Omron CX-Programmer project NewProject (CX-Programmer 9.61)

# PLC traficlight: CP1E N30

## Global symbols (name address type ; comment)
0.00 BOOL  ; STOP
0.01 BOOL  ; START
0.02 BOOL  ; WAKTU 2
0.05 BOOL  ; SENSOR 1
0.06 BOOL  ; SENSOR 2
100.00 BOOL  ; LAMPU MERAH
100.01 BOOL  ; LAMPU KUNING
100.02 BOOL  ; LAMPU HIJAU
100.03 BOOL  ; LAMPU HIJAU
100.04 BOOL  ; LAMPU KUNING
100.05 BOOL  ; LAMPU MERAH
100.06 BOOL  ; IF
5.00 BOOL  ; IR
5.01 BOOL  ; SENSOR
T001 BOOL  ; WAKTU 1
T002 BOOL  ; WAKTU 2
T003 BOOL  ; WAKTU 3
T004 BOOL  ; WAKTU 4
T005 BOOL  ; WAKTU 5
T006 BOOL  ; WAKTU 2
T007 BOOL  ; WAKTU 6

## Program NewProgram1 (cyclic task 0)
Local symbols
END BOOL
SENSOR BOOL

### Section Section1

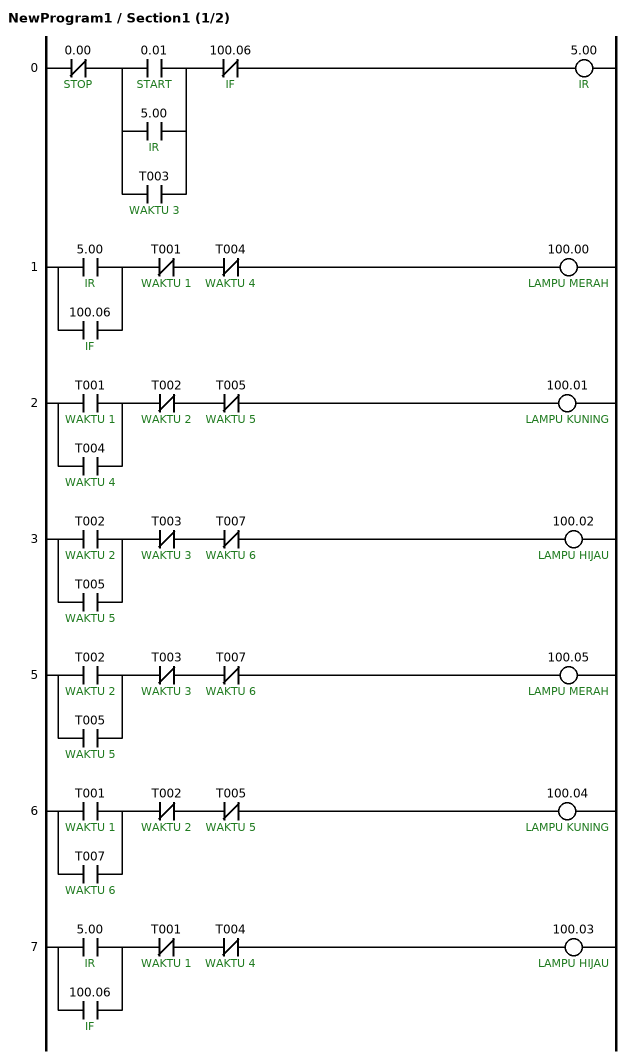
; rung 0
LDNOT 0.00  ; STOP
LD 0.01  ; START
OR 5.00  ; IR
OR T003  ; WAKTU 3
ANDLD
ANDNOT 100.06  ; IF
OUT 5.00  ; IR
; rung 1
LD 5.00  ; IR
OR 100.06  ; IF
ANDNOT T001  ; WAKTU 1
ANDNOT T004  ; WAKTU 4
OUT 100.00  ; LAMPU MERAH
; rung 2
LD T001  ; WAKTU 1
OR T004  ; WAKTU 4
ANDNOT T002  ; WAKTU 2
ANDNOT T005  ; WAKTU 5
OUT 100.01  ; LAMPU KUNING
; rung 3
LD T002  ; WAKTU 2
OR T005  ; WAKTU 5
ANDNOT T003  ; WAKTU 3
ANDNOT T007  ; WAKTU 6
OUT 100.02  ; LAMPU HIJAU
; rung 5
LD T002  ; WAKTU 2
OR T005  ; WAKTU 5
ANDNOT T003  ; WAKTU 3
ANDNOT T007  ; WAKTU 6
OUT 100.05  ; LAMPU MERAH
; rung 6
LD T001  ; WAKTU 1
OR T007  ; WAKTU 6
ANDNOT T002  ; WAKTU 2
ANDNOT T005  ; WAKTU 5
OUT 100.04  ; LAMPU KUNING
; rung 7
LD 5.00  ; IR
OR 100.06  ; IF
ANDNOT T001  ; WAKTU 1
ANDNOT T004  ; WAKTU 4
OUT 100.03  ; LAMPU HIJAU

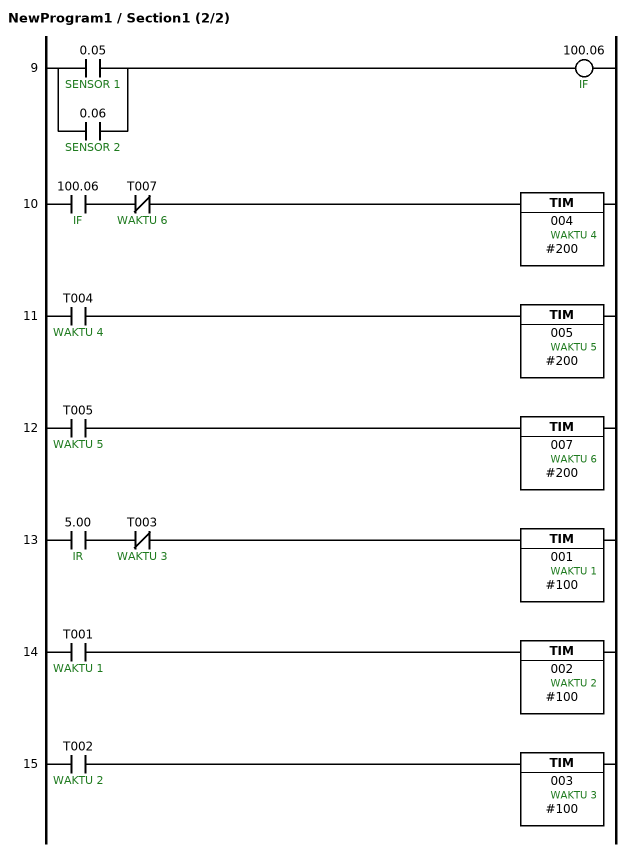
; rung 9
LD 0.05  ; SENSOR 1
OR 0.06  ; SENSOR 2
OUT 100.06  ; IF
; rung 10
LD 100.06  ; IF
ANDNOT T007  ; WAKTU 6
TIM 004 #200  ; WAKTU 4
; rung 11
LD T004  ; WAKTU 4
TIM 005 #200  ; WAKTU 5
; rung 12
LD T005  ; WAKTU 5
TIM 007 #200  ; WAKTU 6
; rung 13
LD 5.00  ; IR
ANDNOT T003  ; WAKTU 3
TIM 001 #100  ; WAKTU 1
; rung 14
LD T001  ; WAKTU 1
TIM 002 #100  ; WAKTU 2
; rung 15
LD T002  ; WAKTU 2
TIM 003 #100  ; WAKTU 3
; rung 16
END(001)

### Section END
; rung 0
END(001)